// Mitsubishi GX Works2 project: 시퀀스 회로 (전후진 제어)   PLC: Q03UDV

PROGRAM MAIN
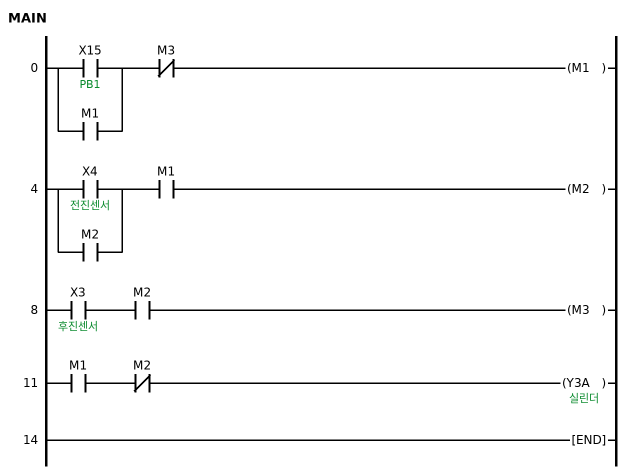
0     LD      X15  ; PB1
      OR      M1
      ANI     M3
      OUT     M1
4     LD      X4  ; 전진센서
      OR      M2
      AND     M1
      OUT     M2
8     LD      X3  ; 후진센서
      AND     M2
      OUT     M3
11    LD      M1
      ANI     M2
      OUT     Y3A  ; 실린더
14    END
END_PROGRAM
